{attribute 'linkalways'} 
{attribute 'no_explicit_call' := 'This FB is a CLASS and must be accessed using methods or properties'}
{attribute 'enable_dynamic_creation'}
FUNCTION_BLOCK Node_F_VN_BitwiseNotImage EXTENDS VisionNode
VAR
    ipSrcImage : _ITcVnImage;
    ipDestImage : _ITcVnImage;
    hrPrev : _HRESULT(S_OK);
	hresult : _HRESULT(S_OK);
END_VAR

METHOD PUBLIC  Clone : I_Node
VAR
	pNode : POINTER TO Node_F_VN_BitwiseNotImage;
END_VAR
pNode := __NEW(Node_F_VN_BitwiseNotImage);
Clone := pNode^;
END_METHOD

METHOD FB_init : BOOL
VAR_INPUT
	bInitRetains : BOOL; // if TRUE, the retain variables are initialized (warm start / cold start)
	bInCopyCode : BOOL;  // if TRUE, the instance afterwards gets moved into the copy code (online change)
END_VAR
AddInput('ipSrcImage', ipSrcImage);
AddInput('hrPrev', hrPrev);
AddOutput('ipDestImage', ipDestImage);
AddOutput('hresult',hresult);
END_METHOD

METHOD PROTECTED OnExecute : HRESULT
hresult.Value := F_VN_BitwiseNotImage(
    ipSrcImage := ipSrcImage.Value,
	ipDestImage := ipDestImage.Value,
	hrPrev:= hrPrev.Value);
END_METHOD

METHOD PUBLIC PreExecutionCheck
VAR_INPUT
	Check : I_PreExecutionChecks;
END_VAR
Check.IsTrue(ipSrcImage.IsValid, 'ipSrcImage must contain an image');
END_METHOD

END_FUNCTION_BLOCK

(* stored: Version 1.1.0.1, ProductVersion 3.1.4024.13
   POU Node_F_VN_BitwiseNotImage: Id {09df121e-16ae-0bee-2400-a7a5c08501dd}, SpecialFunc None
   Folder Constructor: Id {8b3edc21-0bf7-0307-0a4a-4c4f3ace4e71}
   Method Clone: Id {e05a4c03-0b7a-02d4-0fe7-941bb7cceae0}
   Method FB_init: Id {7645416d-852c-0868-28ae-565402097b4e}
   Method OnExecute: Id {5281fcc6-d84f-0a8e-3285-c40253894125}
   Method PreExecutionCheck: Id {069fef0a-6a08-000f-3247-5532e32b1d11} *)
